// TIA Portal V17 export
// export: Created 2025-03-12T15:36:19.2562892Z, ExportSetting WithDefaults, DisplayName Totally Integrated Automation Portal, DisplayVersion V17 Update 8, DisplayName TIA Portal Openness, DisplayVersion V17 Update 8, DisplayName TIA Portal Version Control Interface, DisplayVersion V17, DisplayName SINAMICS Startdrive Advanced, DisplayVersion V17 SP2, DisplayName SINAMICS Startdrive G110M, G120, G120C, G120D, G120P, G115D, DisplayVersion V17 SP2, DisplayName SINAMICS Startdrive G130, G150, S120, S150, SINAMICS MV, S210, DisplayVersion V17 SP2, DisplayName STEP 7 Professional, DisplayVersion V17 Update 8, DisplayName SINUMERIK ONE STEP 7 Toolbox, DisplayVersion V17 Update 12, DisplayName SINUMERIK 840D sl STEP 7 Toolbox, DisplayVersion V17 Update 12, DisplayName STEP 7 Safety, DisplayVersion V17 Update 6, DisplayName WinCC Advanced, DisplayVersion V17 Update 8
DATA_BLOCK "DB16000_OPC_UA_TRIGGER_ALARM"   // DB16000
{ S7_Optimized_Access := 'FALSE' }
VERSION : 0.1
// stored: AutoNumber false, DBAccessibleFromOPCUA true, DBAccessibleFromWebserver true, IsOnlyStoredInLoadMemory false, IsWriteProtectedInAS false
   VAR RETAIN
      CLIENT : Struct
         U01_STA3_MEAS : Struct
            TRIGGERS : Struct
               START_MEAS_NOOZLE : Bool;   // UNIT 01 STATION 3 MEASURING START MEASURING NOOZLE SURFACE DISTANCE TRIGGER
               START_MEAS_NOOZLE_P : Bool;   // UNIT 01 STATION 3 MEASURING START MEASURING NOOZLE SURFACE DISTANCE TRIGGER PULSE
               START_MEAS_LAYER : Bool;   // UNIT 01 STATION 3 MEASURING START MEASURING LAYER THICKNESS TRIGGER
               START_MEAS_LAYER_P : Bool;   // UNIT 01 STATION 3 MEASURING START MEASURING LAYER THICKNESS TRIGGER PULSE
               STOP_MEAS_LAYER : Bool;   // UNIT 01 STATION 3 MEASURING STOP MEASURING LAYER THICKNESS TRIGGER
               STOP_MEAS_LAYER_P : Bool;   // UNIT 01 STATION 3 MEASURING STOP MEASURING LAYER THICKNESS TRIGGER PULSE
               START_CALIBRATION : Bool;   // UNIT 01 STATION 3 MEASURING START CALIBRATING TRIGGER
               START_CALIBRATION_P : Bool;   // UNIT 01 STATION 3 MEASURING START CALIBRATING TRIGGER PULSE
               RESET_PC : Bool;   // UNIT 01 STATION 3 MEASURING RESET PC TRIGGER
               RESET_PC_P : Bool;   // UNIT 01 STATION 3 MEASURING RESET PC TRIGGER PULSE
               READ_VARS : Bool;   // UNIT 01 STATION 3 MEASURING READ VARIABLES TRIGGER
               READ_VARS_P : Bool;   // UNIT 01 STATION 3 MEASURING READ VARIABLES TRIGGER PULSE
            END_STRUCT;
            ALARMS : Struct
               MEAS_NOOZLE_CONNECTION_A : Bool;   // UNIT 01 STATION 3 MEASURING MEASURING NOOZLE SURFACE DISTANCE METHOD CONNECTION ALARM
               MEAS_NOOZLE_METHOD_WORKING_BLOCKED_A : Bool;   // UNIT 01 STATION 3 MEASURING MEASURING NOOZLE SURFACE DISTANCE METHOD WORKING OR BLOCKED ALARM
               MEAS_START_LAYER_CONNECTION_A : Bool;   // UNIT 01 STATION 3 MEASURING START MEASURING LAYER THICKNESS METHOD CONNECTION ALARM
               MEAS_START_LAYER_METHOD_WORKING_BLOCKED_A : Bool;   // UNIT 01 STATION 3 MEASURING START MEASURING LAYER THICKNESS METHOD WORKING OR BLOCKED ALARM
               MEAS_STOP_LAYER_CONNECTION_A : Bool;   // UNIT 01 STATION 3 MEASURING STOP MEASURING LAYER THICKNESS METHOD CONNECTION ALARM
               MEAS_STOP_LAYER_METHOD_WORKING_BLOCKED_A : Bool;   // UNIT 01 STATION 3 MEASURING STOP MEASURING LAYER THICKNESS METHOD WORKING OR BLOCKED ALARM
               CALIBRATE_CONNECTION_A : Bool;   // UNIT 01 STATION 3 MEASURING CALIBRATING METHOD CONNECTION ALARM
               CALIBRATE_METHOD_WORKING_BLOCKED_A : Bool;   // UNIT 01 STATION 3 MEASURING CALIBRATING METHOD WORKING OR BLOCKED ALARM
               RESET_CONNECTION_A : Bool;   // UNIT 01 STATION 3 MEASURING RESET METHOD CONNECTION ALARM
               RESET_METHOD_WORKING_BLOCKED_A : Bool;   // UNIT 01 STATION 3 MEASURING RESET METHOD WORKING OR BLOCKED ALARM
               READ_VAR_CONNECTION_A : Bool;   // UNIT 01 STATION 3 MEASURING READ VARIABLES CONNECTION ALARM
               READ_VAR_METHOD_WORKING_BLOCKED_A : Bool;   // UNIT 01 STATION 3 MEASURING READ VARIABLES WORKING OR BLOCKED ALARM
               PROFILER_CONFIG_A : Bool;   // UNIT 01 STATION 3 MEASURING PROFILER CONFIGURATION ALARM
               ANALYZER_CONFIG_A : Bool;   // UNIT 01 STATION 3 MEASURING ANALYZER CONFIGURATION ALARM
               DMC_STRUCTURE_A : Bool;   // UNIT 01 STATION 3 MEASURING DMC STRUCTURE ALARM
               ACQUISITION_A : Bool;   // UNIT 01 STATION 3 MEASURING ACQUISITON ALARM
               PROFILER_INIT_A : Bool;   // UNIT 01 STATION 3 MEASURING PROFILER INITIALIZTION ALARM
               DISTANCE_CALCULATION_A : Bool;   // UNIT 01 STATION 3 MEASURING DISTANCE CALCULATION ALARM
               LAYER_GROWTH_A : Bool;   // UNIT 01 STATION 3 MEASURING LAYER GROWTH ANALYSIS ALARM
               STORAGE_A : Bool;   // UNIT 01 STATION 3 MEASURING STORAGE ERROR ALARM
               DATABASE_CONNECTION_A : Bool;   // UNIT 01 STATION 3 MEASURING DATABASE CONNECTION ALARM
               CALIBRATION_MISSING_FIX_1_A : Bool;   // UNIT 01 STATION 3 MEASURING MISSING CALIBRATION IN FIXTURE 1 ALARM
               CALIBRATION_MISSING_FIX_2_A : Bool;   // UNIT 01 STATION 3 MEASURING MISSING CALIBRATION IN FIXTURE 2 ALARM
               CALIBRATION_MISSING_FIX_3_A : Bool;   // UNIT 01 STATION 3 MEASURING MISSING CALIBRATION IN FIXTURE 3 ALARM
               CALIBRATION_MISSING_FIX_4_A : Bool;   // UNIT 01 STATION 3 MEASURING MISSING CALIBRATION IN FIXTURE 4 ALARM
               CALIBRATION_OUT_RANGE_FIX_1_A : Bool;   // UNIT 01 STATION 3 MEASURING LAST CALIBRATION OUT OF RANGE IN FIXTURE 1 ALARM
               CALIBRATION_OUT_RANGE_FIX_2_A : Bool;   // UNIT 01 STATION 3 MEASURING LAST CALIBRATION OUT OF RANGE IN FIXTURE 2 ALARM
               CALIBRATION_OUT_RANGE_FIX_3_A : Bool;   // UNIT 01 STATION 3 MEASURING LAST CALIBRATION OUT OF RANGE IN FIXTURE 3 ALARM
               CALIBRATION_OUT_RANGE_FIX_4_A : Bool;   // UNIT 01 STATION 3 MEASURING LAST CALIBRATION OUT OF RANGE IN FIXTURE 4 ALARM
               CALIBRATION_PROC_A : Bool;   // UNIT 01 STATION 3 MEASURING CALIBRATION PROCEDURE ALARM
               MEAS_NOOZLE_DISTANCE_ALARM : Bool;   // UNIT 01 STATION 3 MEASURING NOOZLE DISTANCE ALARM
            END_STRUCT;
            PULSE : Struct
               "1" : Bool;
               "2" : Bool;
               "3" : Bool;
            END_STRUCT;
         END_STRUCT;
         U01_STA3_COAXIAL : Struct
            TRIGGERS : Struct
               START_CAM_CALIBRATION : Bool;   // UNIT 01 STATION 3 COAXIAL CAMERA START CALIBRATION TRIGGER
               START_CAM_CALIBRATION_P : Bool;   // UNIT 01 STATION 3 COAXIAL CAMERA START CALIBRATION TRIGGER PULSE
               START_CAM_ALIGNMENT : Bool;   // UNIT 01 STATION 3 COAXIAL CAMERA START CAPSULE ALIGNMENT TRIGGER
               START_CAM_ALIGNMENT_P : Bool;   // UNIT 01 STATION 3 COAXIAL CAMERA START CAPSULE ALIGNMENT TRIGGER PULSE
               START_CAM_JET_ANALISIS : Bool;   // UNIT 01 STATION 3 COAXIAL CAMERA START JET ANALISIS TRIGGER
               START_CAM_JET_ANALISIS_P : Bool;   // UNIT 01 STATION 3 COAXIAL CAMERA START JET ANALISIS TRIGGER PULSE
               START_CAM_CLADD_ANALISIS : Bool;   // UNIT 01 STATION 3 COAXIAL CAMERA START CLADDING ANALISIS TRIGGER
               START_CAM_CLADD_ANALISIS_P : Bool;   // UNIT 01 STATION 3 COAXIAL CAMERA START CLADDING ANALISIS TRIGGER PULSE
               STOP_CAM_METHODS : Bool;   // UNIT 01 STATION 3 COAXIAL CAMERA STOP SETUP METTHODS TRIGGER
               STOP_CAM_METHODS_P : Bool;   // UNIT 01 STATION 3 COAXIAL CAMERA STOP SETUP METTHODS TRIGGER PULSE
               RESET_PC : Bool;   // UNIT 01 STATION 3 COAXIAL CAMERA RESET PC TRIGGER
               RESET_PC_P : Bool;   // UNIT 01 STATION 3 COAXIAL CAMERA RESET PC TRIGGER PULSE
               READ_VARS : Bool;   // UNIT 01 STATION 3 COAXIAL CAMERA READ VARIABLES TRIGGER
               READ_VARS_P : Bool;   // UNIT 01 STATION 3 COAXIAL CAMERA READ VARIABLES TRIGGER PULSE
            END_STRUCT;
            ALARMS : Struct
               CAM_START_CALIBRATION_CONNECTION_A : Bool;   // UNIT 01 STATION 3 COAXIAL CAMERA START CALIBRATION METHOD CONNECTION ALARM
               CAM_START_CALIBRATION_METHOD_WORKING_BLOCKED_A : Bool;   // UNIT 01 STATION 3 COAXIAL CAMERA START CALIBRATION METHOD WORKING OR BLOCKED ALARM
               CAM_START_ALIGNMENT_CONNECTION_A : Bool;   // UNIT 01 STATION 3 COAXIAL CAMERA START ALIGNMENT METHOD CONNECTION ALARM
               CAM_START_ALIGNMENT_METHOD_WORKING_BLOCKED_A : Bool;   // UNIT 01 STATION 3 COAXIAL CAMERA START ALIGNMENT METHOD WORKING OR BLOCKED ALARM
               CAM_START_JET_ANALISIS_CONNECTION_A : Bool;   // UNIT 01 STATION 3 COAXIAL CAMERA START JET ANALISIS METHOD CONNECTION ALARM
               CAM_START_JET_ANALISIS_METHOD_WORKING_BLOCKED_A : Bool;   // UNIT 01 STATION 3 COAXIAL CAMERA START JET ANALISIS METHOD WORKING OR BLOCKED ALARM
               CAM_START_CLADD_ANALISIS_CONNECTION_A : Bool;   // UNIT 01 STATION 3 COAXIAL CAMERA START CLADDING ANALISIS METHOD CONNECTION ALARM
               CAM_START_CLADD_ANALISIS_METHOD_WORKING_BLOCKED_A : Bool;   // UNIT 01 STATION 3 COAXIAL CAMERA START CLADDING ANALISIS METHOD WORKING OR BLOCKED ALARM
               CAM_STOP_SETUP_METHODS_CONNECTION_A : Bool;   // UNIT 01 STATION 3 COAXIAL CAMERA STOP SETUP METHODS CONNECTION ALARM
               CAM_STOP_SETUP_METHODS_METHOD_WORKING_BLOCKED_A : Bool;   // UNIT 01 STATION 3 COAXIAL CAMERA STOP SETUP METHODS METHOD WORKING OR BLOCKED ALARM
               RESET_PC_CONNECTION_A : Bool;   // UNIT 01 STATION 3 COAXIAL CAMERA REST PC METHOD CONNECTION ALARM
               RESET_PC_METHOD_WORKING_BLOCKED_A : Bool;   // UNIT 01 STATION 3 COAXIAL CAMERA REST PC METHOD WORKING OR BLOCKED ALARM
               READ_VARS_CONNECTION_A : Bool;   // UNIT 01 STATION 3 COAXIAL CAMERA READ VARIABLES METHOD CONNECTION ALARM
               READ_VARS_METHOD_WORKING_BLOCKED_A : Bool;   // UNIT 01 STATION 3 COAXIAL CAMERA READ VARIABLES METHOD WORKING BLOCKED ALARM
               CAMERA_FAILED_A : Bool;   // UNIT 01 STATION 3 COAXIAL CAMERA FAILED ALARM
               NO_LIGHT_A : Bool;   // UNIT 01 STATION 3 COAXIAL CAMERA NO LIGHT ALARM
               CAPSULE_MISALIGNED_A : Bool;   // UNIT 01 STATION 3 COAXIAL CAMERA CAPSULE MISALIGNED ALARM
               JET_FAILED_ALARM : Bool;   // UNIT 01 STATION 3 COAXIAL CAMERA JET FAILED ALARM
               NO_POWDER_A : Bool;   // UNIT 01 STATION 3 COAXIAL CAMERA NO POWDER ALARM
               LASER_MISALIGNED_A : Bool;   // UNIT 01 STATION 3 COAXIAL CAMERA LASER MISALIGNED ALARM
               DIRTY_CAPSULE_A : Bool;   // UNIT 01 STATION 3 COAXIAL CAMERA DIRTY CAPSULE ALARM
               DMC_STRUCTURE_A : Bool;   // UNIT 01 STATION 3 COAXIAL CAMERA DMC STRUCTURE ALARM
            END_STRUCT;
         END_STRUCT;
         U02_STA2_MEAS : Struct
            TRIGGERS : Struct
               START_MEAS : Bool;   // UNIT 02 STATION 2 MEASURING START MEASURING TRIGGER
               START_MEAS_P : Bool;   // UNIT 02 STATION 2 MEASURING START MEASURING TRIGGER PULSE
               START_CALIBRATION : Bool;   // UNIT 02 STATION 2 MEASURING START CALIBRATING TRIGGER
               START_CALIBRATION_P : Bool;   // UNIT 02 STATION 2 MEASURING START CALIBRATING TRIGGER PULSE
               RESET_PC : Bool;   // UNIT 02 STATION 2 MEASURING RESET PC TRIGGER
               RESET_PC_P : Bool;   // UNIT 02 STATION 2 MEASURING RESET PC TRIGGER PULSE
               READ_VARS : Bool;   // UNIT 02 STATION 2 MEASURING READ VARIABLES TRIGGER
               READ_VARS_P : Bool;   // UNIT 02 STATION 2 MEASURING READ VARIABLES TRIGGER PULSE
            END_STRUCT;
            ALARMS : Struct
               MEAS_CONNECTION_A : Bool;   // UNIT 02 STATION 2 MEASURING MEASURING METHOD CONNECTION ALARM
               MEAS_METHOD_WORKING_BLOCKED_A : Bool;   // UNIT 02 STATION 2 MEASURING MEASURING METHOD WORKING OR BLOCKED ALARM
               CALIBRATE_CONNECTION_A : Bool;   // UNIT 02 STATION 2 MEASURING CALIBRATING METHOD CONNECTION ALARM
               CALIBRATE_METHOD_WORKING_BLOCKED_A : Bool;   // UNIT 02 STATION 2 MEASURING CALIBRATING METHOD WORKING OR BLOCKED ALARM
               RESET_CONNECTION_A : Bool;   // UNIT 02 STATION 2 MEASURING RESET METHOD CONNECTION ALARM
               RESET_METHOD_WORKING_BLOCKED_A : Bool;   // UNIT 02 STATION 2 MEASURING RESET METHOD WORKING OR BLOCKED ALARM
               READ_VAR_CONNECTION_A : Bool;   // UNIT 02 STATION 2 MEASURING READ VARIABLES CONNECTION ALARM
               READ_VAR_METHOD_WORKING_BLOCKED_A : Bool;   // UNIT 02 STATION 2 MEASURING READ VARIABLES WORKING OR BLOCKED ALARM
               PROFILER_CONFIG_A : Bool;   // UNIT 02 STATION 2 MEASURING PROFILER CONFIGURATION ALARM
               ANALYZER_CONFIG_A : Bool;   // UNIT 02 STATION 2 MEASURING ANALYZER CONFIGURATION ALARM
               DMC_STRUCTURE_A : Bool;   // UNIT 02 STATION 2 MEASURING DMC STRUCTURE ALARM
               ACQUISITION_A : Bool;   // UNIT 02 STATION 2 MEASURING ACQUISITON ALARM
               PROFILER_INIT_A : Bool;   // UNIT 02 STATION 2 MEASURING PROFILER INITIALIZTION ALARM
               UMBRELLA_A : Bool;   // UNIT 02 STATION 2 MEASURING UMBRELLA ANALYSIS ALARM
               RUNOUT_A : Bool;   // UNIT 02 STATION 2 MEASURING RUN OUT ANALYSIS ALARM
               LAYER_GROWTH_A : Bool;   // UNIT 02 STATION 2 MEASURING LAYER GROWTH ANALYSIS ALARM
               SURFACE_DEFECTS_A : Bool;   // UNIT 02 STATION 2 MEASURING SURFACE DEFECTS ANALYSIS ALARM
               STORAGE_A : Bool;   // UNIT 02 STATION 2 MEASURING STORAGE ERROR ALARM
               DATABASE_CONNECTION_A : Bool;   // UNIT 02 STATION 2 MEASURING DATABASE CONNECTION ALARM
               CALIBRATION_MISSING_FIX_1_A : Bool;   // UNIT 02 STATION 2 MEASURING MISSING CALIBRATION IN FIXTURE 1 ALARM
               CALIBRATION_MISSING_FIX_2_A : Bool;   // UNIT 02 STATION 2 MEASURING MISSING CALIBRATION IN FIXTURE 2 ALARM
               CALIBRATION_MISSING_FIX_3_A : Bool;   // UNIT 02 STATION 2 MEASURING MISSING CALIBRATION IN FIXTURE 3 ALARM
               CALIBRATION_MISSING_FIX_4_A : Bool;   // UNIT 02 STATION 2 MEASURING MISSING CALIBRATION IN FIXTURE 4 ALARM
               CALIBRATION_OUT_RANGE_FIX_1_A : Bool;   // UNIT 02 STATION 2 MEASURING LAST CALIBRATION OUT OF RANGE IN FIXTURE 1 ALARM
               CALIBRATION_OUT_RANGE_FIX_2_A : Bool;   // UNIT 02 STATION 2 MEASURING LAST CALIBRATION OUT OF RANGE IN FIXTURE 2 ALARM
               CALIBRATION_OUT_RANGE_FIX_3_A : Bool;   // UNIT 02 STATION 2 MEASURING LAST CALIBRATION OUT OF RANGE IN FIXTURE 3 ALARM
               CALIBRATION_OUT_RANGE_FIX_4_A : Bool;   // UNIT 02 STATION 2 MEASURING LAST CALIBRATION OUT OF RANGE IN FIXTURE 4 ALARM
               CALIBRATION_PROC_A : Bool;   // UNIT 02 STATION 2 MEASURING CALIBRATION PROCEDURE ALARM
            END_STRUCT;
            PULSE : Struct
               "1" : Bool;
            END_STRUCT;
         END_STRUCT;
         U02_STA3_MEAS : Struct
            TRIGGERS : Struct
               START_MEAS_NOOZLE : Bool;   // UNIT 02 STATION 3 MEASURING START MEASURING NOOZLE SURFACE DISTANCE TRIGGER
               START_MEAS_NOOZLE_P : Bool;   // UNIT 02 STATION 3 MEASURING START MEASURING NOOZLE SURFACE DISTANCE TRIGGER PULSE
               START_MEAS_LAYER : Bool;   // UNIT 02 STATION 3 MEASURING START MEASURING LAYER THICKNESS TRIGGER
               START_MEAS_LAYER_P : Bool;   // UNIT 02 STATION 3 MEASURING START MEASURING LAYER THICKNESS TRIGGER PULSE
               STOP_MEAS_LAYER : Bool;   // UNIT 02 STATION 3 MEASURING STOP MEASURING LAYER THICKNESS TRIGGER
               STOP_MEAS_LAYER_P : Bool;   // UNIT 02 STATION 3 MEASURING STOP MEASURING LAYER THICKNESS TRIGGER PULSE
               START_CALIBRATION : Bool;   // UNIT 02 STATION 3 MEASURING START CALIBRATING TRIGGER
               START_CALIBRATION_P : Bool;   // UNIT 02 STATION 3 MEASURING START CALIBRATING TRIGGER PULSE
               RESET_PC : Bool;   // UNIT 02 STATION 3 MEASURING RESET PC TRIGGER
               RESET_PC_P : Bool;   // UNIT 02 STATION 3 MEASURING RESET PC TRIGGER PULSE
               READ_VARS : Bool;   // UNIT 02 STATION 3 MEASURING READ VARIABLES TRIGGER
               READ_VARS_P : Bool;   // UNIT 02 STATION 3 MEASURING READ VARIABLES TRIGGER PULSE
            END_STRUCT;
            ALARMS : Struct
               MEAS_NOOZLE_CONNECTION_A : Bool;   // UNIT 02 STATION 3 MEASURING MEASURING NOOZLE SURFACE DISTANCE METHOD CONNECTION ALARM
               MEAS_NOOZLE_METHOD_WORKING_BLOCKED_A : Bool;   // UNIT 02 STATION 3 MEASURING MEASURING NOOZLE SURFACE DISTANCE METHOD WORKING OR BLOCKED ALARM
               MEAS_START_LAYER_CONNECTION_A : Bool;   // UNIT 02 STATION 3 MEASURING START MEASURING LAYER THICKNESS METHOD CONNECTION ALARM
               MEAS_START_LAYER_METHOD_WORKING_BLOCKED_A : Bool;   // UNIT 02 STATION 3 MEASURING START MEASURING LAYER THICKNESS METHOD WORKING OR BLOCKED ALARM
               MEAS_STOP_LAYER_CONNECTION_A : Bool;   // UNIT 02 STATION 3 MEASURING STOP MEASURING LAYER THICKNESS METHOD CONNECTION ALARM
               MEAS_STOP_LAYER_METHOD_WORKING_BLOCKED_A : Bool;   // UNIT 02 STATION 3 MEASURING STOP MEASURING LAYER THICKNESS METHOD WORKING OR BLOCKED ALARM
               CALIBRATE_CONNECTION_A : Bool;   // UNIT 02 STATION 3 MEASURING CALIBRATING METHOD CONNECTION ALARM
               CALIBRATE_METHOD_WORKING_BLOCKED_A : Bool;   // UNIT 02 STATION 3 MEASURING CALIBRATING METHOD WORKING OR BLOCKED ALARM
               RESET_CONNECTION_A : Bool;   // UNIT 02 STATION 3 MEASURING RESET METHOD CONNECTION ALARM
               RESET_METHOD_WORKING_BLOCKED_A : Bool;   // UNIT 02 STATION 3 MEASURING RESET METHOD WORKING OR BLOCKED ALARM
               READ_VAR_CONNECTION_A : Bool;   // UNIT 02 STATION 3 MEASURING READ VARIABLES CONNECTION ALARM
               READ_VAR_METHOD_WORKING_BLOCKED_A : Bool;   // UNIT 02 STATION 3 MEASURING READ VARIABLES WORKING OR BLOCKED ALARM
               PROFILER_CONFIG_A : Bool;   // UNIT 02 STATION 3 MEASURING PROFILER CONFIGURATION ALARM
               ANALYZER_CONFIG_A : Bool;   // UNIT 02 STATION 3 MEASURING ANALYZER CONFIGURATION ALARM
               DMC_STRUCTURE_A : Bool;   // UNIT 02 STATION 3 MEASURING DMC STRUCTURE ALARM
               ACQUISITION_A : Bool;   // UNIT 02 STATION 3 MEASURING ACQUISITON ALARM
               PROFILER_INIT_A : Bool;   // UNIT 02 STATION 3 MEASURING PROFILER INITIALIZTION ALARM
               DISTANCE_CALCULATION_A : Bool;   // UNIT 02 STATION 3 MEASURING DISTANCE CALCULATION ALARM
               LAYER_GROWTH_A : Bool;   // UNIT 02 STATION 3 MEASURING LAYER GROWTH ANALYSIS ALARM
               STORAGE_A : Bool;   // UNIT 02 STATION 3 MEASURING STORAGE ERROR ALARM
               DATABASE_CONNECTION_A : Bool;   // UNIT 02 STATION 3 MEASURING DATABASE CONNECTION ALARM
               CALIBRATION_MISSING_FIX_1_A : Bool;   // UNIT 02 STATION 3 MEASURING MISSING CALIBRATION IN FIXTURE 1 ALARM
               CALIBRATION_MISSING_FIX_2_A : Bool;   // UNIT 02 STATION 3 MEASURING MISSING CALIBRATION IN FIXTURE 2 ALARM
               CALIBRATION_MISSING_FIX_3_A : Bool;   // UNIT 02 STATION 3 MEASURING MISSING CALIBRATION IN FIXTURE 3 ALARM
               CALIBRATION_MISSING_FIX_4_A : Bool;   // UNIT 02 STATION 3 MEASURING MISSING CALIBRATION IN FIXTURE 4 ALARM
               CALIBRATION_OUT_RANGE_FIX_1_A : Bool;   // UNIT 02 STATION 3 MEASURING LAST CALIBRATION OUT OF RANGE IN FIXTURE 1 ALARM
               CALIBRATION_OUT_RANGE_FIX_2_A : Bool;   // UNIT 02 STATION 3 MEASURING LAST CALIBRATION OUT OF RANGE IN FIXTURE 2 ALARM
               CALIBRATION_OUT_RANGE_FIX_3_A : Bool;   // UNIT 02 STATION 3 MEASURING LAST CALIBRATION OUT OF RANGE IN FIXTURE 3 ALARM
               CALIBRATION_OUT_RANGE_FIX_4_A : Bool;   // UNIT 02 STATION 3 MEASURING LAST CALIBRATION OUT OF RANGE IN FIXTURE 4 ALARM
               CALIBRATION_PROC_A : Bool;   // UNIT 02 STATION 3 MEASURING CALIBRATION PROCEDURE ALARM
               MEAS_NOOZLE_DISTANCE_ALARM : Bool;   // UNIT 02 STATION 3 MEASURING NOOZLE DISTANCE ALARM
            END_STRUCT;
            PULSE : Struct
               "1" : Bool;
               "2" : Bool;
               "3" : Bool;
            END_STRUCT;
         END_STRUCT;
         U02_STA3_COAXIAL : Struct
            TRIGGERS : Struct
               START_CAM_CALIBRATION : Bool;   // UNIT 02 STATION 3 COAXIAL CAMERA START CALIBRATION TRIGGER
               START_CAM_CALIBRATION_P : Bool;   // UNIT 02 STATION 3 COAXIAL CAMERA START CALIBRATION TRIGGER PULSE
               START_CAM_ALIGNMENT : Bool;   // UNIT 02 STATION 3 COAXIAL CAMERA START CAPSULE ALIGNMENT TRIGGER
               START_CAM_ALIGNMENT_P : Bool;   // UNIT 02 STATION 3 COAXIAL CAMERA START CAPSULE ALIGNMENT TRIGGER PULSE
               START_CAM_JET_ANALISIS : Bool;   // UNIT 02 STATION 3 COAXIAL CAMERA START JET ANALISIS TRIGGER
               START_CAM_JET_ANALISIS_P : Bool;   // UNIT 02 STATION 3 COAXIAL CAMERA START JET ANALISIS TRIGGER PULSE
               START_CAM_CLADD_ANALISIS : Bool;   // UNIT 02 STATION 3 COAXIAL CAMERA START CLADDING ANALISIS TRIGGER
               START_CAM_CLADD_ANALISIS_P : Bool;   // UNIT 02 STATION 3 COAXIAL CAMERA START CLADDING ANALISIS TRIGGER PULSE
               STOP_CAM_METHODS : Bool;   // UNIT 02 STATION 3 COAXIAL CAMERA STOP SETUP METTHODS TRIGGER
               STOP_CAM_METHODS_P : Bool;   // UNIT 02 STATION 3 COAXIAL CAMERA STOP SETUP METTHODS TRIGGER PULSE
               RESET_PC : Bool;   // UNIT 02 STATION 3 COAXIAL CAMERA RESET PC TRIGGER
               RESET_PC_P : Bool;   // UNIT 02 STATION 3 COAXIAL CAMERA RESET PC TRIGGER PULSE
               READ_VARS : Bool;   // UNIT 02 STATION 3 COAXIAL CAMERA READ VARIABLES TRIGGER
               READ_VARS_P : Bool;   // UNIT 02 STATION 3 COAXIAL CAMERA READ VARIABLES TRIGGER PULSE
            END_STRUCT;
            ALARMS : Struct
               CAM_START_CALIBRATION_CONNECTION_A : Bool;   // UNIT 02 STATION 3 COAXIAL CAMERA START CALIBRATION METHOD CONNECTION ALARM
               CAM_START_CALIBRATION_METHOD_WORKING_BLOCKED_A : Bool;   // UNIT 02 STATION 3 COAXIAL CAMERA START CALIBRATION METHOD WORKING OR BLOCKED ALARM
               CAM_START_ALIGNMENT_CONNECTION_A : Bool;   // UNIT 02 STATION 3 COAXIAL CAMERA START ALIGNMENT METHOD CONNECTION ALARM
               CAM_START_ALIGNMENT_METHOD_WORKING_BLOCKED_A : Bool;   // UNIT 02 STATION 3 COAXIAL CAMERA START ALIGNMENT METHOD WORKING OR BLOCKED ALARM
               CAM_START_JET_ANALISIS_CONNECTION_A : Bool;   // UNIT 02 STATION 3 COAXIAL CAMERA START JET ANALISIS METHOD CONNECTION ALARM
               CAM_START_JET_ANALISIS_METHOD_WORKING_BLOCKED_A : Bool;   // UNIT 02 STATION 3 COAXIAL CAMERA START JET ANALISIS METHOD WORKING OR BLOCKED ALARM
               CAM_START_CLADD_ANALISIS_CONNECTION_A : Bool;   // UNIT 02 STATION 3 COAXIAL CAMERA START CLADDING ANALISIS METHOD CONNECTION ALARM
               CAM_START_CLADD_ANALISIS_METHOD_WORKING_BLOCKED_A : Bool;   // UNIT 02 STATION 3 COAXIAL CAMERA START CLADDING ANALISIS METHOD WORKING OR BLOCKED ALARM
               CAM_STOP_SETUP_METHODS_CONNECTION_A : Bool;   // UNIT 02 STATION 3 COAXIAL CAMERA STOP SETUP METHODS CONNECTION ALARM
               CAM_STOP_SETUP_METHODS_METHOD_WORKING_BLOCKED_A : Bool;   // UNIT 02 STATION 3 COAXIAL CAMERA STOP SETUP METHODS METHOD WORKING OR BLOCKED ALARM
               RESET_PC_CONNECTION_A : Bool;   // UNIT 02 STATION 3 COAXIAL CAMERA REST PC METHOD CONNECTION ALARM
               RESET_PC_METHOD_WORKING_BLOCKED_A : Bool;   // UNIT 02 STATION 3 COAXIAL CAMERA REST PC METHOD WORKING OR BLOCKED ALARM
               READ_VARS_CONNECTION_A : Bool;   // UNIT 02 STATION 3 COAXIAL CAMERA READ VARIABLES METHOD CONNECTION ALARM
               READ_VARS_METHOD_WORKING_BLOCKED_A : Bool;   // UNIT 02 STATION 3 COAXIAL CAMERA READ VARIABLES METHOD WORKING BLOCKED ALARM
               CAMERA_FAILED_A : Bool;   // UNIT 02 STATION 3 COAXIAL CAMERA FAILED ALARM
               NO_LIGHT_A : Bool;   // UNIT 02 STATION 3 COAXIAL CAMERA NO LIGHT ALARM
               CAPSULE_MISALIGNED_A : Bool;   // UNIT 02 STATION 3 COAXIAL CAMERA CAPSULE MISALIGNED ALARM
               JET_FAILED_ALARM : Bool;   // UNIT 02 STATION 3 COAXIAL CAMERA JET FAILED ALARM
               NO_POWDER_A : Bool;   // UNIT 02 STATION 3 COAXIAL CAMERA NO POWDER ALARM
               LASER_MISALIGNED_A : Bool;   // UNIT 02 STATION 3 COAXIAL CAMERA LASER MISALIGNED ALARM
               DIRTY_CAPSULE_A : Bool;   // UNIT 02 STATION 3 COAXIAL CAMERA DIRTY CAPSULE ALARM
               DMC_STRUCTURE_A : Bool;   // UNIT 02 STATION 3 COAXIAL CAMERA DMC STRUCTURE ALARM
            END_STRUCT;
         END_STRUCT;
         U03_MEAS_STA_MEAS_A : Struct
            TRIGGERS : Struct
               START_MEAS : Bool;   // UNIT 03 MEASURING STATION FACE A START MEASURING TRIGGER
               START_MEAS_P : Bool;   // UNIT 03 MEASURING STATION FACE A START MEASURING TRIGGER PULSE
               START_CALIBRATION : Bool;   // UNIT 03 MEASURING STATION FACE A START CALIBRATING TRIGGER
               START_CALIBRATION_P : Bool;   // UNIT 03 MEASURING STATION FACE A START CALIBRATING TRIGGER PULSE
               RESET_PC : Bool;   // UNIT 03 MEASURING STATION FACE A RESET PC TRIGGER
               RESET_PC_P : Bool;   // UNIT 03 MEASURING STATION FACE A RESET PC TRIGGER PULSE
               READ_VARS : Bool;   // UNIT 03 MEASURING STATION FACE A READ VARIABLES TRIGGER
               READ_VARS_P : Bool;   // UNIT 03 MEASURING STATION FACE A READ VARIABLES TRIGGER PULSE
            END_STRUCT;
            ALARMS : Struct
               MEAS_CONNECTION_A : Bool;   // UNIT 03 MEASURING STATION FACE A MEASURING METHOD CONNECTION ALARM
               MEAS_METHOD_WORKING_BLOCKED_A : Bool;   // UNIT 03 MEASURING STATION FACE A MEASURING METHOD WORKING OR BLOCKED ALARM
               CALIBRATE_CONNECTION_A : Bool;   // UNIT 03 MEASURING STATION FACE A CALIBRATING METHOD CONNECTION ALARM
               CALIBRATE_METHOD_WORKING_BLOCKED_A : Bool;   // UNIT 03 MEASURING STATION FACE A CALIBRATING METHOD WORKING OR BLOCKED ALARM
               RESET_CONNECTION_A : Bool;   // UNIT 03 MEASURING STATION FACE A RESET METHOD CONNECTION ALARM
               RESET_METHOD_WORKING_BLOCKED_A : Bool;   // UNIT 03 MEASURING STATION FACE A RESET METHOD WORKING OR BLOCKED ALARM
               READ_VAR_CONNECTION_A : Bool;   // UNIT 03 MEASURING STATION FACE A READ VARIABLES CONNECTION ALARM
               READ_VAR_METHOD_WORKING_BLOCKED_A : Bool;   // UNIT 03 MEASURING STATION FACE A READ VARIABLES WORKING OR BLOCKED ALARM
               PROFILER_CONFIG_A : Bool;   // UNIT 03 MEASURING STATION FACE A PROFILER CONFIGURATION ALARM
               ANALYZER_CONFIG_A : Bool;   // UNIT 03 MEASURING STATION FACE A ANALYZER CONFIGURATION ALARM
               DMC_STRUCTURE_A : Bool;   // UNIT 03 MEASURING STATION FACE A DMC STRUCTURE ALARM
               ACQUISITION_A : Bool;   // UNIT 03 MEASURING STATION FACE A ACQUISITON ALARM
               PROFILER_INIT_A : Bool;   // UNIT 03 MEASURING STATION FACE A PROFILER INITIALIZTION ALARM
               UMBRELLA_A : Bool;   // UNIT 03 MEASURING STATION FACE A UMBRELLA ANALYSIS ALARM
               RUNOUT_A : Bool;   // UNIT 03 MEASURING STATION FACE A RUN OUT ANALYSIS ALARM
               DISTANCE_CALCULATION_A : Bool;   // UNIT 03 MEASURING STATION FACE A DISTANCE CALCULATION ALARM
               LAYER_GROWTH_A : Bool;   // UNIT 03 MEASURING STATION FACE A LAYER GROWTH ANALYSIS ALARM
               SURFACE_DEFECTS_A : Bool;   // UNIT 03 MEASURING STATION FACE A SURFACE DEFECTS ANALYSIS ALARM
               STORAGE_A : Bool;   // UNIT 03 MEASURING STATION FACE A STORAGE ERROR ALARM
               DATABASE_CONNECTION_A : Bool;   // UNIT 03 MEASURING STATION FACE A DATABASE CONNECTION ALARM
               CALIBRATION_MISSING_A : Bool;   // UNIT 03 MEASURING STATION FACE A MISSING CALIBRATION ALARM
               CALIBRATION_PROC_A : Bool;   // UNIT 03 MEASURING STATION FACE A CALIBRATION PROCEDURE ALARM
            END_STRUCT;
            PULSE : Struct
               "1" : Bool;
            END_STRUCT;
         END_STRUCT;
         U03_MEAS_STA_MEAS_B : Struct
            TRIGGERS : Struct
               START_MEAS : Bool;   // UNIT 03 MEASURING STATION FACE B START MEASURING TRIGGER
               START_MEAS_P : Bool;   // UNIT 03 MEASURING STATION FACE B START MEASURING TRIGGER PULSE
               START_CALIBRATION : Bool;   // UNIT 03 MEASURING STATION FACE B START CALIBRATING TRIGGER
               START_CALIBRATION_P : Bool;   // UNIT 03 MEASURING STATION FACE B START CALIBRATING TRIGGER PULSE
               RESET_PC : Bool;   // UNIT 03 MEASURING STATION FACE B RESET PC TRIGGER
               RESET_PC_P : Bool;   // UNIT 03 MEASURING STATION FACE B RESET PC TRIGGER PULSE
               READ_VARS : Bool;   // UNIT 03 MEASURING STATION FACE A READ VARIABLES TRIGGER
               READ_VARS_P : Bool;   // UNIT 03 MEASURING STATION FACE A READ VARIABLES TRIGGER PULSE
            END_STRUCT;
            ALARMS : Struct
               MEAS_CONNECTION_A : Bool;   // UNIT 03 MEASURING STATION FACE B MEASURING METHOD CONNECTION ALARM
               MEAS_METHOD_WORKING_BLOCKED_A : Bool;   // UNIT 03 MEASURING STATION FACE B MEASURING METHOD WORKING OR BLOCKED ALARM
               CALIBRATE_CONNECTION_A : Bool;   // UNIT 03 MEASURING STATION FACE B CALIBRATING METHOD CONNECTION ALARM
               CALIBRATE_METHOD_WORKING_BLOCKED_A : Bool;   // UNIT 03 MEASURING STATION FACE B CALIBRATING METHOD WORKING OR BLOCKED ALARM
               RESET_CONNECTION_A : Bool;   // UNIT 03 MEASURING STATION FACE B RESET METHOD CONNECTION ALARM
               RESET_METHOD_WORKING_BLOCKED_A : Bool;   // UNIT 03 MEASURING STATION FACE B RESET METHOD WORKING OR BLOCKED ALARM
               READ_VAR_CONNECTION_A : Bool;   // UNIT 03 MEASURING STATION FACE B READ VARIABLES CONNECTION ALARM
               READ_VAR_METHOD_WORKING_BLOCKED_A : Bool;   // UNIT 03 MEASURING STATION FACE B READ VARIABLES WORKING OR BLOCKED ALARM
               PROFILER_CONFIG_A : Bool;   // UNIT 03 MEASURING STATION FACE B PROFILER CONFIGURATION ALARM
               ANALYZER_CONFIG_A : Bool;   // UNIT 03 MEASURING STATION FACE B ANALYZER CONFIGURATION ALARM
               DMC_STRUCTURE_A : Bool;   // UNIT 03 MEASURING STATION FACE B DMC STRUCTURE ALARM
               ACQUISITION_A : Bool;   // UNIT 03 MEASURING STATION FACE B ACQUISITON ALARM
               PROFILER_INIT_A : Bool;   // UNIT 03 MEASURING STATION FACE B PROFILER INITIALIZTION ALARM
               UMBRELLA_A : Bool;   // UNIT 03 MEASURING STATION FACE B UMBRELLA ANALYSIS ALARM
               RUNOUT_A : Bool;   // UNIT 03 MEASURING STATION FACE B RUN OUT ANALYSIS ALARM
               DISTANCE_CALCULATION_A : Bool;   // UNIT 03 MEASURING STATION FACE B DISTANCE CALCULATION ALARM
               LAYER_GROWTH_A : Bool;   // UNIT 03 MEASURING STATION FACE B LAYER GROWTH ANALYSIS ALARM
               SURFACE_DEFECTS_A : Bool;   // UNIT 03 MEASURING STATION FACE B SURFACE DEFECTS ANALYSIS ALARM
               STORAGE_A : Bool;   // UNIT 03 MEASURING STATION FACE B STORAGE ERROR ALARM
               DATABASE_CONNECTION_A : Bool;   // UNIT 03 MEASURING STATION FACE B DATABASE CONNECTION ALARM
               CALIBRATION_MISSING_A : Bool;   // UNIT 03 MEASURING STATION FACE B MISSING CALIBRATION ALARM
               CALIBRATION_PROC_A : Bool;   // UNIT 03 MEASURING STATION FACE B CALIBRATION PROCEDURE ALARM
            END_STRUCT;
            PULSE : Struct
               "1" : Bool;
            END_STRUCT;
         END_STRUCT;
      END_STRUCT;
      MASTER : Struct
         SPARE : Bool;
      END_STRUCT;
   END_VAR
BEGIN
END_DATA_BLOCK
